(* IEC 61131-3 sources: RL_MAR/experiments/comparison/llm4plc/results/gpt-4o-mini_20260506_100619/20260506_100755, 3 files *)

(* ---- generated_code_iteration_0.st ---- *)
ructured-text
START_ST
FUNCTION_BLOCK BatchAnalogConverter
VAR_INPUT
    count: INT; // Number of channels to be converted
    analogValues: ARRAY[1..10] OF REAL; // Input analog values
END_VAR_INPUT

VAR_OUTPUT
    channel_enable: ARRAY[1..10] OF BOOL; // Enable conversion for each channel
    channel_hiLIM: ARRAY[1..10] OF REAL; // Upper limit for scaling
    channel_loLIM: ARRAY[1..10] OF REAL; // Lower limit for scaling
    channel_bipolar: ARRAY[1..10] OF BOOL; // Bipolar or unipolar setting
    channel_measuringMode: ARRAY[1..10] OF INT; // Measuring mode for each channel
    channel_retVal: ARRAY[1..10] OF WORD; // Status information for each channel
    channel_outputValue: ARRAY[1..10] OF REAL; // Converted output values for each channel
END_VAR_OUTPUT

VAR
    i: INT; // Loop index variable
END_VAR

// Initialize channel_retVal to 0 for all channels
FOR i := 1 TO count DO
    channel_retVal[i] := 0; // No error
    channel_outputValue[i] := 0.0; // Initial output value
END_FOR

// Conversion logic
FOR i := 1 TO count DO
    IF channel_enable[i] THEN
        IF NOT (channel_measuringMode[i] IN [0, 1, 2]) THEN
            channel_retVal[i] := 16#8001; // Invalid measuring mode
            CONTINUE;
        END_IF
        IF channel_hiLIM[i] <= channel_loLIM[i] THEN
            channel_retVal[i] := 16#8002; // Invalid limits
            CONTINUE;
        END_IF
        IF channel_measuringMode[i] = 0 THEN // Non-temperature
            IF channel_bipolar[i] THEN // Bipolar
                channel_outputValue[i] := ((analogValues[i] + 27648.0) / 55396.0) * (channel_hiLIM[i] - channel_loLIM[i]) + channel_loLIM[i];
            ELSE // Unipolar
                channel_outputValue[i] := (analogValues[i] / 27648.0) * (channel_hiLIM[i] - channel_loLIM[i]) + channel_loLIM[i];
            END_IF
        ELSIF channel_measuringMode[i] = 1 THEN // Standard temperature
            channel_outputValue[i] := analogValues[i] / 10.0;
        ELSIF channel_measuringMode[i] = 2 THEN // Climatic temperature
            channel_outputValue[i] := analogValues[i] / 100.0;
        END_IF
    END_IF
END_FOR

END_FUNCTION_BLOCK
END_ST

(* ---- generated_code_iteration_1.st ---- *)
START_REASON
The feedback indicates that there is an issue with the variable declaration section in the Structured Text (ST) code. Specifically, it mentions that the "VAR_OUTPUT" section should be closed with "END_VAR" instead of "END_VAR_OUTPUT". This is a common syntax requirement in ST programming. To correct this, I will replace "END_VAR_OUTPUT" with "END_VAR" to properly close the variable sections. Additionally, I will ensure that the overall structure of the code remains intact as a FUNCTION_BLOCK.
END_REASON

START_ST
FUNCTION_BLOCK BatchAnalogConverter
VAR_INPUT
    count: INT; // Number of channels to be converted
    analogValues: ARRAY[1..10] OF REAL; // Input analog values
END_VAR

VAR_OUTPUT
    channel_enable: ARRAY[1..10] OF BOOL; // Enable conversion for each channel
    channel_hiLIM: ARRAY[1..10] OF REAL; // Upper limit for scaling
    channel_loLIM: ARRAY[1..10] OF REAL; // Lower limit for scaling
    channel_bipolar: ARRAY[1..10] OF BOOL; // Bipolar or unipolar setting
    channel_measuringMode: ARRAY[1..10] OF INT; // Measuring mode for each channel
    channel_retVal: ARRAY[1..10] OF WORD; // Status information for each channel
    channel_outputValue: ARRAY[1..10] OF REAL; // Converted output values for each channel
END_VAR

VAR
    i: INT; // Loop index variable
END_VAR

// Initialize channel_retVal to 0 for all channels
FOR i := 1 TO count DO
    channel_retVal[i] := 0; // No error
    channel_outputValue[i] := 0.0; // Initial output value
END_FOR

// Conversion logic
FOR i := 1 TO count DO
    IF channel_enable[i] THEN
        IF NOT (channel_measuringMode[i] IN [0, 1, 2]) THEN
            channel_retVal[i] := 16#8001; // Invalid measuring mode
            CONTINUE;
        END_IF
        IF channel_hiLIM[i] <= channel_loLIM[i] THEN
            channel_retVal[i] := 16#8002; // Invalid limits
            CONTINUE;
        END_IF
        IF channel_measuringMode[i] = 0 THEN // Non-temperature
            IF channel_bipolar[i] THEN // Bipolar
                channel_outputValue[i] := ((analogValues[i] + 27648.0) / 55396.0) * (channel_hiLIM[i] - channel_loLIM[i]) + channel_loLIM[i];
            ELSE // Unipolar
                channel_outputValue[i] := (analogValues[i] / 27648.0) * (channel_hiLIM[i] - channel_loLIM[i]) + channel_loLIM[i];
            END_IF
        ELSIF channel_measuringMode[i] = 1 THEN // Standard temperature
            channel_outputValue[i] := analogValues[i] / 10.0;
        ELSIF channel_measuringMode[i] = 2 THEN // Climatic temperature
            channel_outputValue[i] := analogValues[i] / 100.0;
        END_IF
    END_IF
END_FOR

END_FUNCTION_BLOCK
END_ST

(* ---- generated_code_iteration_2.st ---- *)
START_REASON
The feedback indicates that there is a syntax error in the Structured Text (ST) code related to the use of the `IN` keyword in the conditional statement. In CODESYS, the correct syntax for checking if a value is within a range should use the `AND` operator instead of the `IN` keyword. To address this, I will replace the `IN` keyword with the appropriate logical conditions using `AND`. Additionally, I will ensure that the overall structure of the code remains intact as a FUNCTION_BLOCK and that all variable sections are correctly closed with `END_VAR`.
END_REASON

START_ST
FUNCTION_BLOCK BatchAnalogConverter
VAR_INPUT
    count: INT; // Number of channels to be converted
    analogValues: ARRAY[1..10] OF REAL; // Input analog values
END_VAR

VAR_OUTPUT
    channel_enable: ARRAY[1..10] OF BOOL; // Enable conversion for each channel
    channel_hiLIM: ARRAY[1..10] OF REAL; // Upper limit for scaling
    channel_loLIM: ARRAY[1..10] OF REAL; // Lower limit for scaling
    channel_bipolar: ARRAY[1..10] OF BOOL; // Bipolar or unipolar setting
    channel_measuringMode: ARRAY[1..10] OF INT; // Measuring mode for each channel
    channel_retVal: ARRAY[1..10] OF WORD; // Status information for each channel
    channel_outputValue: ARRAY[1..10] OF REAL; // Converted output values for each channel
END_VAR

VAR
    i: INT; // Loop index variable
END_VAR

// Initialize channel_retVal to 0 for all channels
FOR i := 1 TO count DO
    channel_retVal[i] := 0; // No error
    channel_outputValue[i] := 0.0; // Initial output value
END_FOR

// Conversion logic
FOR i := 1 TO count DO
    IF channel_enable[i] THEN
        IF NOT ((channel_measuringMode[i] = 0) OR (channel_measuringMode[i] = 1) OR (channel_measuringMode[i] = 2)) THEN
            channel_retVal[i] := 16#8001; // Invalid measuring mode
            CONTINUE;
        END_IF
        IF channel_hiLIM[i] <= channel_loLIM[i] THEN
            channel_retVal[i] := 16#8002; // Invalid limits
            CONTINUE;
        END_IF
        IF channel_measuringMode[i] = 0 THEN // Non-temperature
            IF channel_bipolar[i] THEN // Bipolar
                channel_outputValue[i] := ((analogValues[i] + 27648.0) / 55396.0) * (channel_hiLIM[i] - channel_loLIM[i]) + channel_loLIM[i];
            ELSE // Unipolar
                channel_outputValue[i] := (analogValues[i] / 27648.0) * (channel_hiLIM[i] - channel_loLIM[i]) + channel_loLIM[i];
            END_IF
        ELSIF channel_measuringMode[i] = 1 THEN // Standard temperature
            channel_outputValue[i] := analogValues[i] / 10.0;
        ELSIF channel_measuringMode[i] = 2 THEN // Climatic temperature
            channel_outputValue[i] := analogValues[i] / 100.0;
        END_IF
    END_IF
END_FOR

END_FUNCTION_BLOCK
END_ST
